//{attribute 'qualified_only'}
VAR_GLOBAL CONSTANT
	MAX_UNIT_NUMBER : BYTE := 9;
//	MIN_UNIT_NUMBER_STRING : STRING := '1';
//	MAX_UNIT_NUMBER_STRING : STRING := BYTE_TO_STRING(MAX_UNIT_NUMBER);
END_VAR

(* stored: Version 1.1.0.1, ProductVersion 3.1.4024.12
   GVL gCONSTANT: Id {4a691510-55c1-4e8d-ac93-7012a8cc4c0a} *)
